FUNCTION_BLOCK Component EXTENDS Composite
VAR
END_VAR

METHOD logStatus
VAR
	sMessage				: STRING;		
END_VAR
// Local status 
SUPER^.logStatus();
END_METHOD

END_FUNCTION_BLOCK

(* stored: Version 1.1.0.1, ProductVersion 3.1.4024.12
   POU Component: Id {c9af56f0-8ee3-4ea4-a4e9-a3e6db04f829}, SpecialFunc None
   Method logStatus: Id {f22a363c-34c3-47a9-bc12-f1fe4d1b2d58} *)
